ABB RAPID module: Wobj_wObj_Teste.mod

MODULE Wobj_wObj_Teste
	! Points are read in order of declaration.
  ! Please do not change the order of points!

  LOCAL PERS robtarget pWobj_U_PointX1:=[[2086.681,-1458.722,319.1031],[0.340816289186478,0.508037865161896,0.777828752994537,-0.1439588367939],[-1,-1,1,0],[9E+09,9E+09,9E+09,9E+09,9E+09,9E+09]];
	LOCAL PERS robtarget pWobj_U_PointX2:=[[1709.912,-1457.474,320.2891],[0.340810239315033,0.508042931556702,0.777827978134155,-0.143959730863571],[-1,-1,0,0],[9E+09,9E+09,9E+09,9E+09,9E+09,9E+09]];
	LOCAL PERS robtarget pWobj_U_PointY1:=[[2087.352,-2053.779,320.0703],[0.340808779001236,0.508042335510254,0.777828812599182,-0.143960565328598],[-1,-1,0,0],[9E+09,9E+09,9E+09,9E+09,9E+09,9E+09]];

ENDMODULE
